// Mitsubishi GX Works2 project: Projec1 (Advance)_FX3U   PLC: FX3U/FX3UC

PROGRAM MAIN
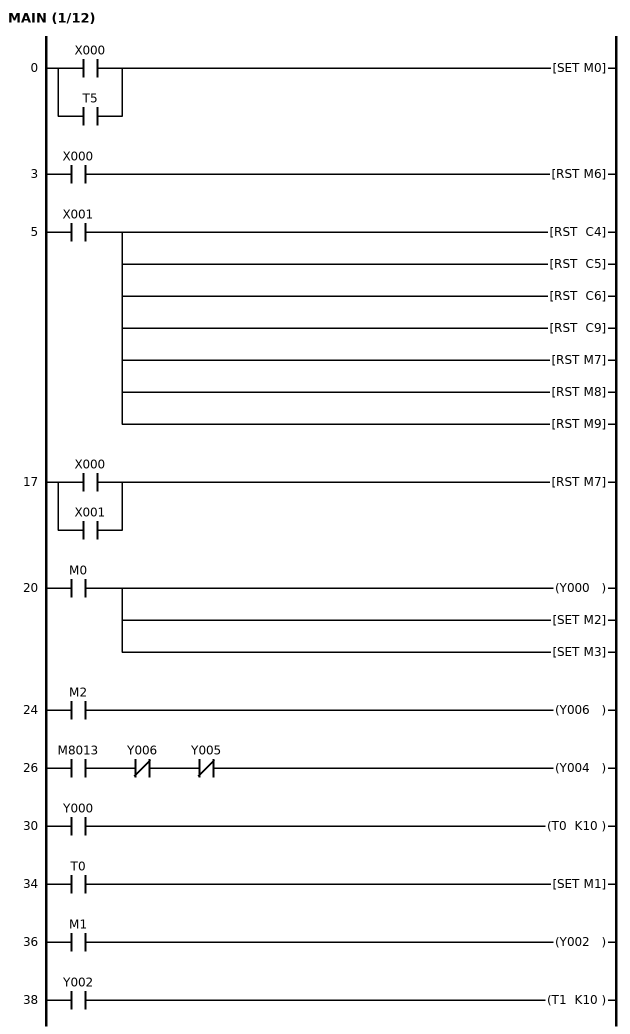
0     LD      X000
      OR      T5
      SET     M0
3     LD      X000
      RST     M6
5     LD      X001
      RST     C4
      RST     C5
      RST     C6
      RST     C9
      RST     M7
      RST     M8
      RST     M9
17    LD      X000
      OR      X001
      RST     M7
20    LD      M0
      OUT     Y000
      SET     M2
      SET     M3
24    LD      M2
      OUT     Y006
26    LD      M8013
      ANI     Y006
      ANI     Y005
      OUT     Y004
30    LD      Y000
      OUT     T0 K10
34    LD      T0
      SET     M1
36    LD      M1
      OUT     Y002
38    LD      Y002
      OUT     T1 K10
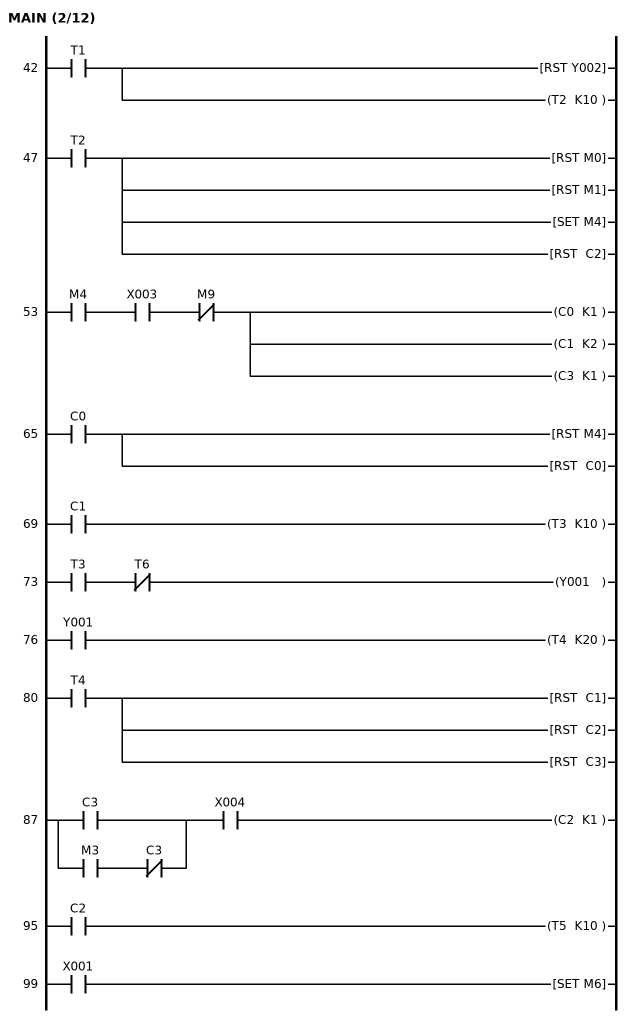
42    LD      T1
      RST     Y002
      OUT     T2 K10
47    LD      T2
      RST     M0
      RST     M1
      SET     M4
      RST     C2
53    LD      M4
      AND     X003
      ANI     M9
      OUT     C0 K1
      OUT     C1 K2
      OUT     C3 K1
65    LD      C0
      RST     M4
      RST     C0
69    LD      C1
      OUT     T3 K10
73    LD      T3
      ANI     T6
      OUT     Y001
76    LD      Y001
      OUT     T4 K20
80    LD      T4
      RST     C1
      RST     C2
      RST     C3
87    LD      C3
      LD      M3
      ANI     C3
      ORB
      AND     X004
      OUT     C2 K1
95    LD      C2
      OUT     T5 K10
99    LD      X001
      SET     M6
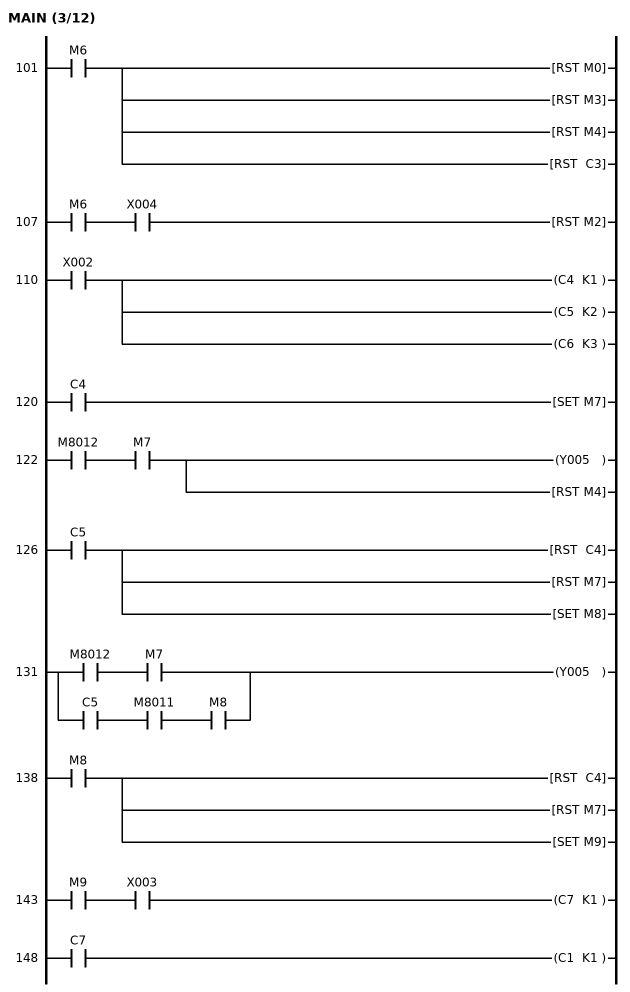
101   LD      M6
      RST     M0
      RST     M3
      RST     M4
      RST     C3
107   LD      M6
      AND     X004
      RST     M2
110   LD      X002
      OUT     C4 K1
      OUT     C5 K2
      OUT     C6 K3
120   LD      C4
      SET     M7
122   LD      M8012
      AND     M7
      OUT     Y005
      RST     M4
126   LD      C5
      RST     C4
      RST     M7
      SET     M8
131   LD      M8012
      AND     M7
      LD      C5
      AND     M8011
      AND     M8
      ORB
      OUT     Y005
138   LD      M8
      RST     C4
      RST     M7
      SET     M9
143   LD      M9
      AND     X003
      OUT     C7 K1
148   LD      C7
      OUT     C1 K1
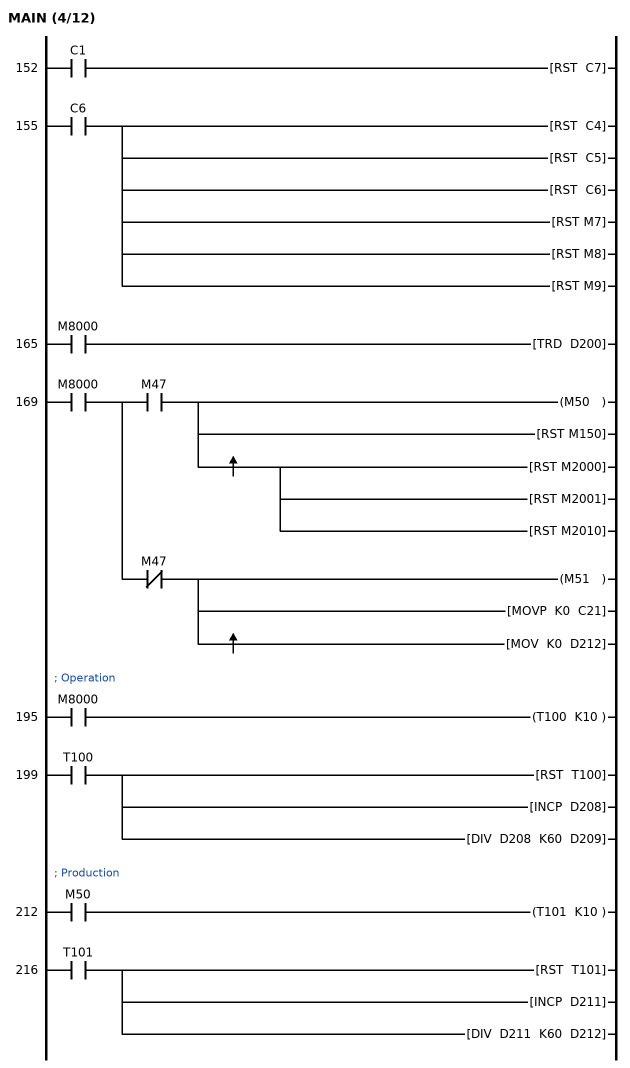
152   LD      C1
      RST     C7
155   LD      C6
      RST     C4
      RST     C5
      RST     C6
      RST     M7
      RST     M8
      RST     M9
165   LD      M8000
      TRD     D200
169   LD      M8000
      MPS
      AND     M47
      OUT     M50
      RST     M150
      MEP
      RST     M2000
      RST     M2001
      RST     M2010
      MPP
      ANI     M47
      OUT     M51
      MOVP    K0 C21
      MEP
      MOV     K0 D212
; Operation
195   LD      M8000
      OUT     T100 K10
199   LD      T100
      RST     T100
      INCP    D208
      DIV     D208 K60 D209
; Production
212   LD      M50
      OUT     T101 K10
216   LD      T101
      RST     T101
      INCP    D211
      DIV     D211 K60 D212
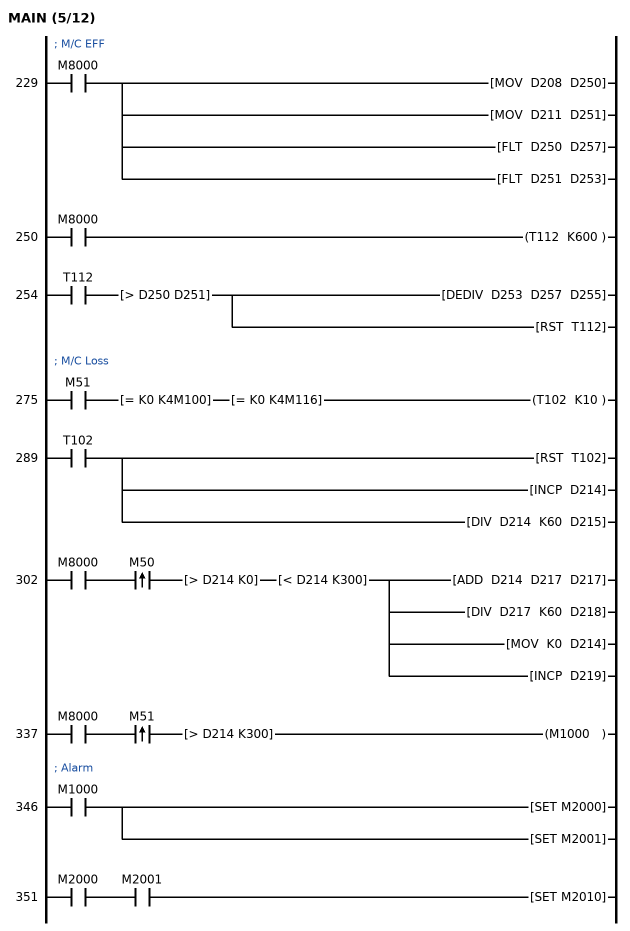
; M/C EFF
229   LD      M8000
      MOV     D208 D250
      MOV     D211 D251
      FLT     D250 D257
      FLT     D251 D253
250   LD      M8000
      OUT     T112 K600
254   LD      T112
      AND>    D250 D251
      DEDIV   D253 D257 D255
      RST     T112
; M/C Loss
275   LD      M51
      AND=    K0 K4M100
      AND=    K0 K4M116
      OUT     T102 K10
289   LD      T102
      RST     T102
      INCP    D214
      DIV     D214 K60 D215
302   LD      M8000
      ANDP    M50
      AND>    D214 K0
      AND<    D214 K300
      ADD     D214 D217 D217
      DIV     D217 K60 D218
      MOV     K0 D214
      INCP    D219
337   LD      M8000
      ANDP    M51
      AND>    D214 K300
      OUT     M1000
; Alarm
346   LD      M1000
      SET     M2000
      SET     M2001
351   LD      M2000
      AND     M2001
      SET     M2010
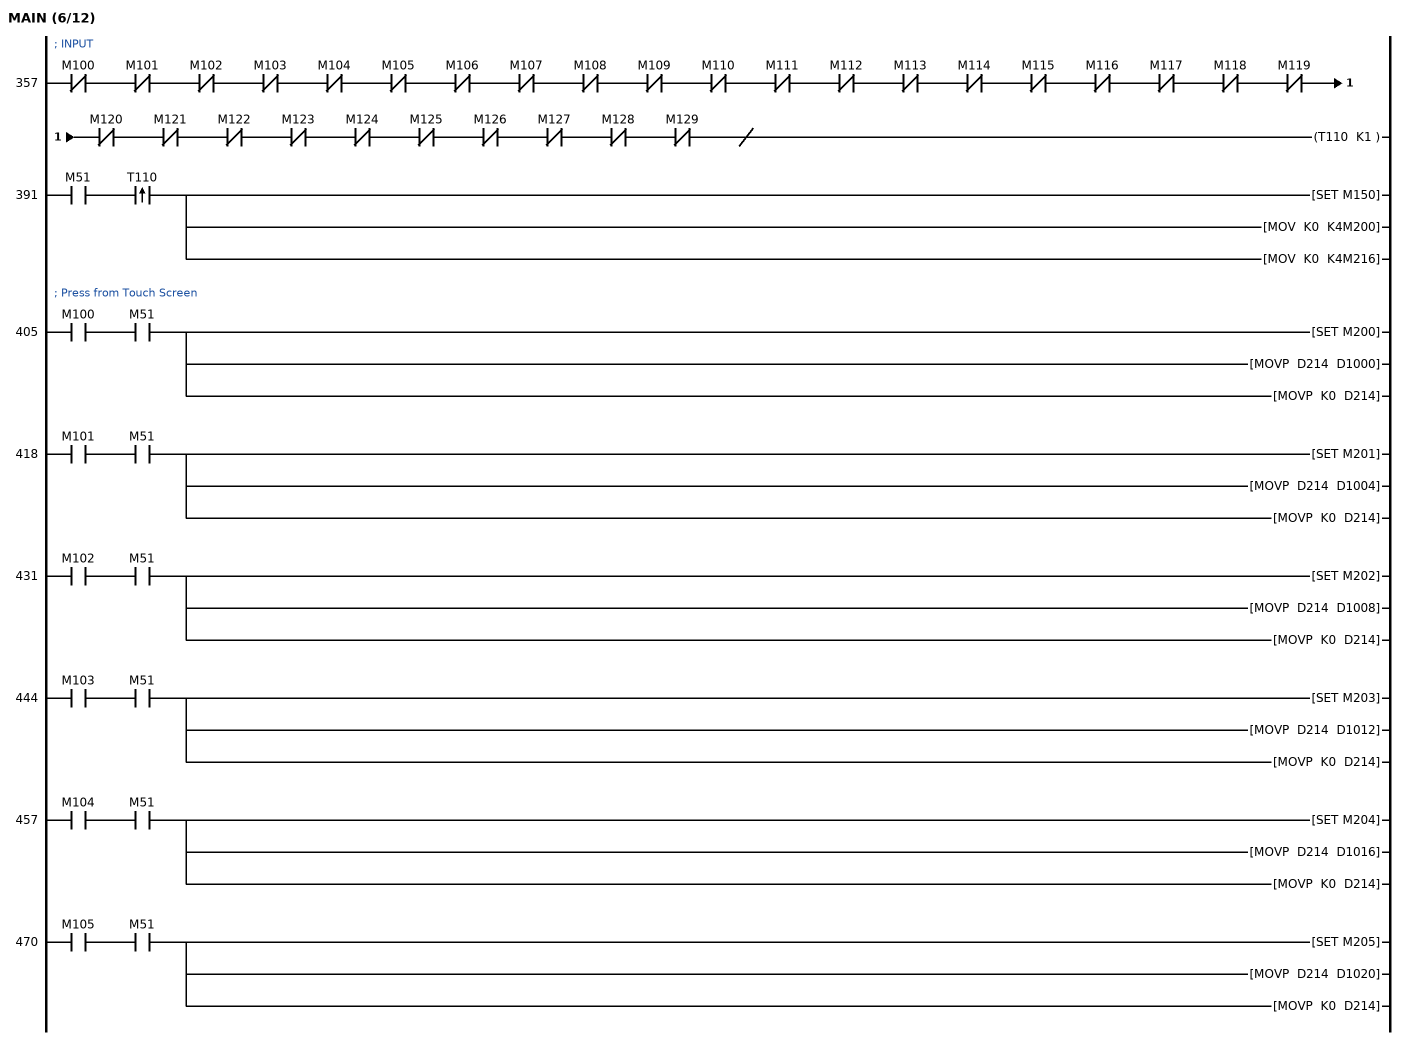
; INPUT
357   LDI     M100
      ANI     M101
      ANI     M102
      ANI     M103
      ANI     M104
      ANI     M105
      ANI     M106
      ANI     M107
      ANI     M108
      ANI     M109
      ANI     M110
      ANI     M111
      ANI     M112
      ANI     M113
      ANI     M114
      ANI     M115
      ANI     M116
      ANI     M117
      ANI     M118
      ANI     M119
      ANI     M120
      ANI     M121
      ANI     M122
      ANI     M123
      ANI     M124
      ANI     M125
      ANI     M126
      ANI     M127
      ANI     M128
      ANI     M129
      INV
      OUT     T110 K1
391   LD      M51
      ANDP    T110
      SET     M150
      MOV     K0 K4M200
      MOV     K0 K4M216
; Press from Touch Screen
405   LD      M100
      AND     M51
      SET     M200
      MOVP    D214 D1000
      MOVP    K0 D214
418   LD      M101
      AND     M51
      SET     M201
      MOVP    D214 D1004
      MOVP    K0 D214
431   LD      M102
      AND     M51
      SET     M202
      MOVP    D214 D1008
      MOVP    K0 D214
444   LD      M103
      AND     M51
      SET     M203
      MOVP    D214 D1012
      MOVP    K0 D214
457   LD      M104
      AND     M51
      SET     M204
      MOVP    D214 D1016
      MOVP    K0 D214
470   LD      M105
      AND     M51
      SET     M205
      MOVP    D214 D1020
      MOVP    K0 D214
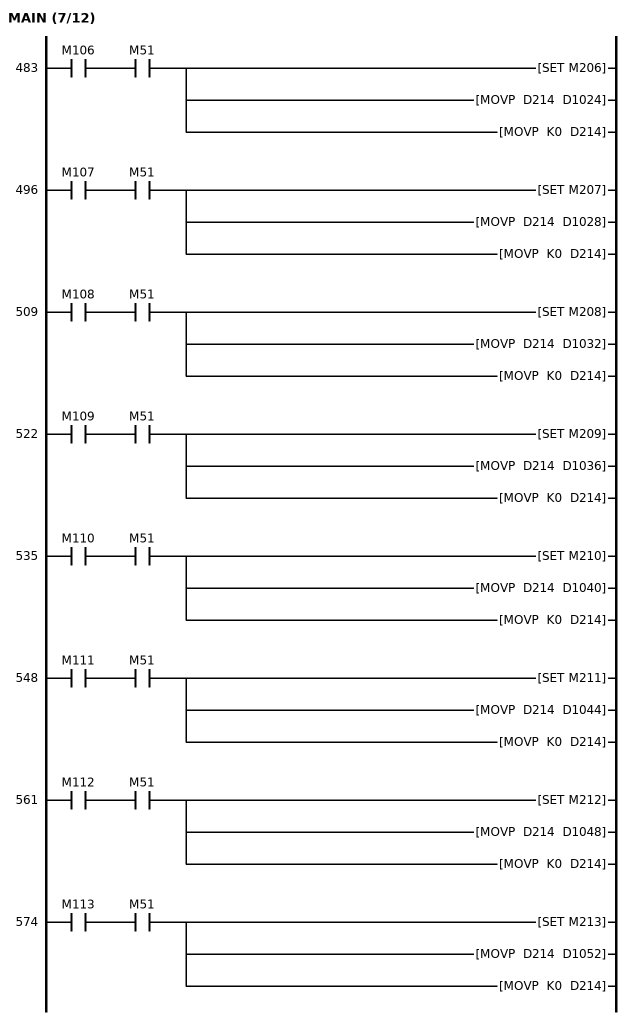
483   LD      M106
      AND     M51
      SET     M206
      MOVP    D214 D1024
      MOVP    K0 D214
496   LD      M107
      AND     M51
      SET     M207
      MOVP    D214 D1028
      MOVP    K0 D214
509   LD      M108
      AND     M51
      SET     M208
      MOVP    D214 D1032
      MOVP    K0 D214
522   LD      M109
      AND     M51
      SET     M209
      MOVP    D214 D1036
      MOVP    K0 D214
535   LD      M110
      AND     M51
      SET     M210
      MOVP    D214 D1040
      MOVP    K0 D214
548   LD      M111
      AND     M51
      SET     M211
      MOVP    D214 D1044
      MOVP    K0 D214
561   LD      M112
      AND     M51
      SET     M212
      MOVP    D214 D1048
      MOVP    K0 D214
574   LD      M113
      AND     M51
      SET     M213
      MOVP    D214 D1052
      MOVP    K0 D214
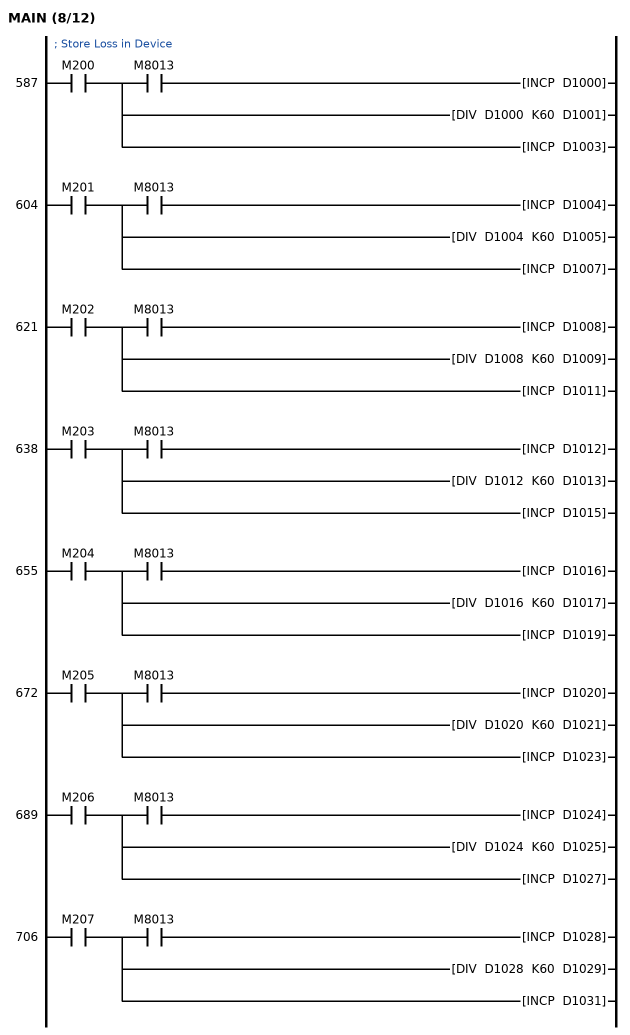
; Store Loss in Device
587   LD      M200
      MPS
      AND     M8013
      INCP    D1000
      MPP
      DIV     D1000 K60 D1001
      INCP    D1003
604   LD      M201
      MPS
      AND     M8013
      INCP    D1004
      MPP
      DIV     D1004 K60 D1005
      INCP    D1007
621   LD      M202
      MPS
      AND     M8013
      INCP    D1008
      MPP
      DIV     D1008 K60 D1009
      INCP    D1011
638   LD      M203
      MPS
      AND     M8013
      INCP    D1012
      MPP
      DIV     D1012 K60 D1013
      INCP    D1015
655   LD      M204
      MPS
      AND     M8013
      INCP    D1016
      MPP
      DIV     D1016 K60 D1017
      INCP    D1019
672   LD      M205
      MPS
      AND     M8013
      INCP    D1020
      MPP
      DIV     D1020 K60 D1021
      INCP    D1023
689   LD      M206
      MPS
      AND     M8013
      INCP    D1024
      MPP
      DIV     D1024 K60 D1025
      INCP    D1027
706   LD      M207
      MPS
      AND     M8013
      INCP    D1028
      MPP
      DIV     D1028 K60 D1029
      INCP    D1031
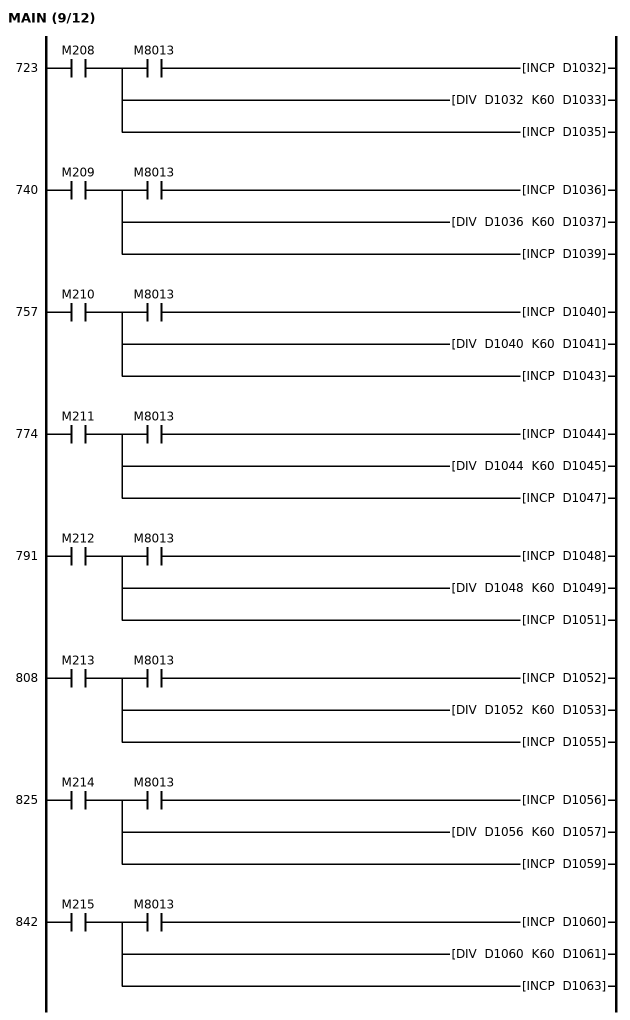
723   LD      M208
      MPS
      AND     M8013
      INCP    D1032
      MPP
      DIV     D1032 K60 D1033
      INCP    D1035
740   LD      M209
      MPS
      AND     M8013
      INCP    D1036
      MPP
      DIV     D1036 K60 D1037
      INCP    D1039
757   LD      M210
      MPS
      AND     M8013
      INCP    D1040
      MPP
      DIV     D1040 K60 D1041
      INCP    D1043
774   LD      M211
      MPS
      AND     M8013
      INCP    D1044
      MPP
      DIV     D1044 K60 D1045
      INCP    D1047
791   LD      M212
      MPS
      AND     M8013
      INCP    D1048
      MPP
      DIV     D1048 K60 D1049
      INCP    D1051
808   LD      M213
      MPS
      AND     M8013
      INCP    D1052
      MPP
      DIV     D1052 K60 D1053
      INCP    D1055
825   LD      M214
      MPS
      AND     M8013
      INCP    D1056
      MPP
      DIV     D1056 K60 D1057
      INCP    D1059
842   LD      M215
      MPS
      AND     M8013
      INCP    D1060
      MPP
      DIV     D1060 K60 D1061
      INCP    D1063
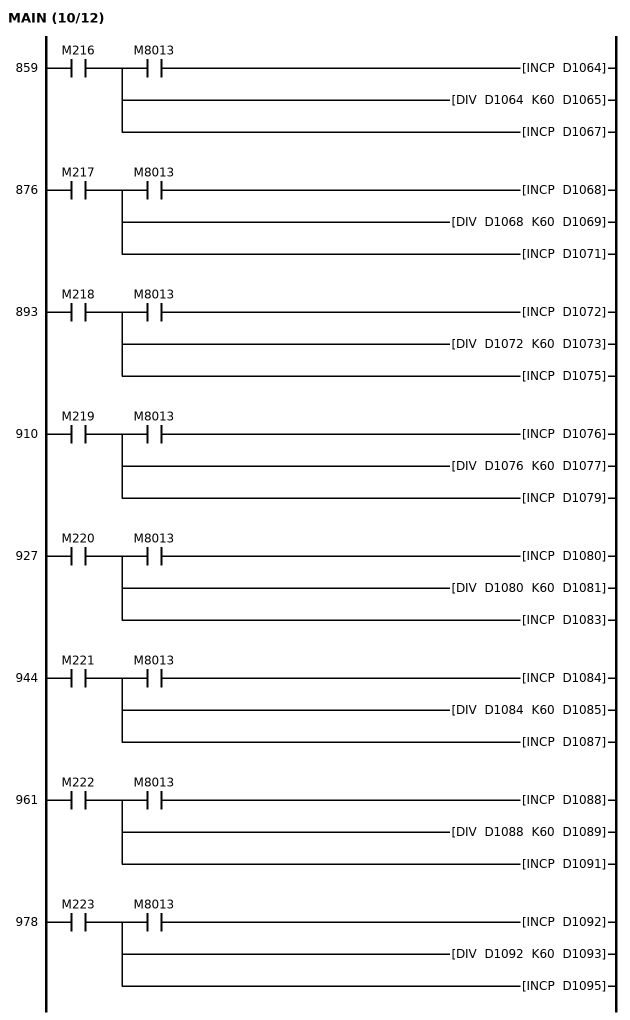
859   LD      M216
      MPS
      AND     M8013
      INCP    D1064
      MPP
      DIV     D1064 K60 D1065
      INCP    D1067
876   LD      M217
      MPS
      AND     M8013
      INCP    D1068
      MPP
      DIV     D1068 K60 D1069
      INCP    D1071
893   LD      M218
      MPS
      AND     M8013
      INCP    D1072
      MPP
      DIV     D1072 K60 D1073
      INCP    D1075
910   LD      M219
      MPS
      AND     M8013
      INCP    D1076
      MPP
      DIV     D1076 K60 D1077
      INCP    D1079
927   LD      M220
      MPS
      AND     M8013
      INCP    D1080
      MPP
      DIV     D1080 K60 D1081
      INCP    D1083
944   LD      M221
      MPS
      AND     M8013
      INCP    D1084
      MPP
      DIV     D1084 K60 D1085
      INCP    D1087
961   LD      M222
      MPS
      AND     M8013
      INCP    D1088
      MPP
      DIV     D1088 K60 D1089
      INCP    D1091
978   LD      M223
      MPS
      AND     M8013
      INCP    D1092
      MPP
      DIV     D1092 K60 D1093
      INCP    D1095
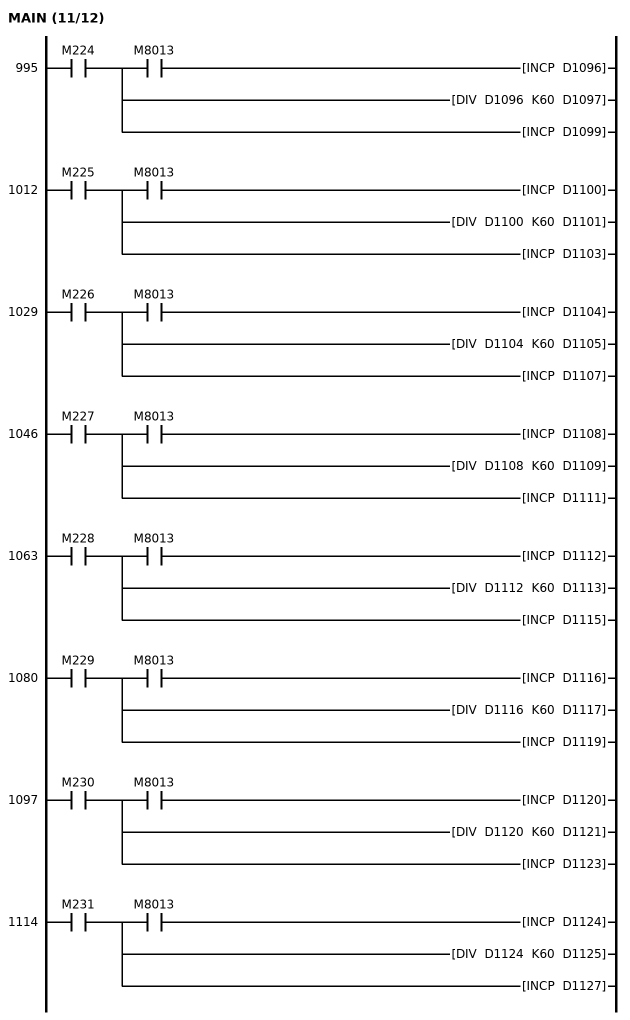
995   LD      M224
      MPS
      AND     M8013
      INCP    D1096
      MPP
      DIV     D1096 K60 D1097
      INCP    D1099
1012  LD      M225
      MPS
      AND     M8013
      INCP    D1100
      MPP
      DIV     D1100 K60 D1101
      INCP    D1103
1029  LD      M226
      MPS
      AND     M8013
      INCP    D1104
      MPP
      DIV     D1104 K60 D1105
      INCP    D1107
1046  LD      M227
      MPS
      AND     M8013
      INCP    D1108
      MPP
      DIV     D1108 K60 D1109
      INCP    D1111
1063  LD      M228
      MPS
      AND     M8013
      INCP    D1112
      MPP
      DIV     D1112 K60 D1113
      INCP    D1115
1080  LD      M229
      MPS
      AND     M8013
      INCP    D1116
      MPP
      DIV     D1116 K60 D1117
      INCP    D1119
1097  LD      M230
      MPS
      AND     M8013
      INCP    D1120
      MPP
      DIV     D1120 K60 D1121
      INCP    D1123
1114  LD      M231
      MPS
      AND     M8013
      INCP    D1124
      MPP
      DIV     D1124 K60 D1125
      INCP    D1127
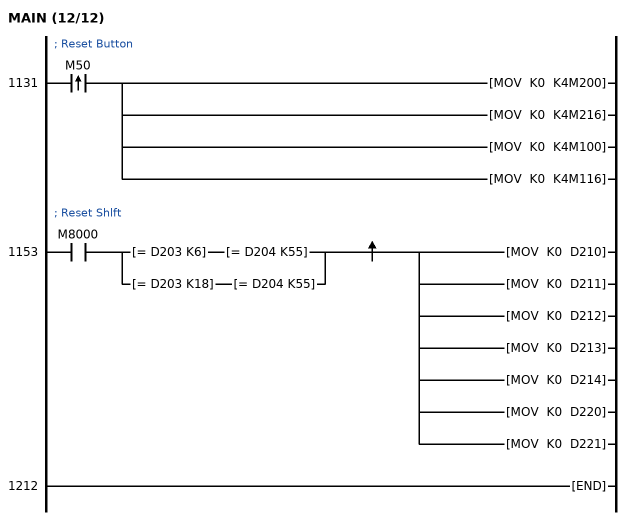
; Reset Button
1131  LDP     M50
      MOV     K0 K4M200
      MOV     K0 K4M216
      MOV     K0 K4M100
      MOV     K0 K4M116
; Reset Shlft
1153  LD      M8000
      LD=     D203 K6
      AND=    D204 K55
      LD=     D203 K18
      AND=    D204 K55
      ORB
      ANB
      MEP
      MOV     K0 D210
      MOV     K0 D211
      MOV     K0 D212
      MOV     K0 D213
      MOV     K0 D214
      MOV     K0 D220
      MOV     K0 D221
1212  END
END_PROGRAM
